(* PLC project Unnamed, Unknown Unnamed 1 *)
(* stored: creationDateTime 2025-10-24T15:36:12, modificationDateTime 2026-02-02T21:17:16 *)

PROGRAM program0
  VAR
    RawADC : INT;
    Temp : INT;
  END_VAR

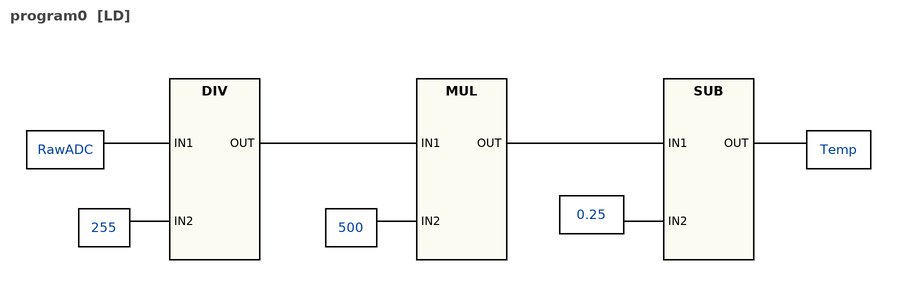
(* LD diagram, written out as Structured Text *)
Temp := RawADC / 255 * 500 - 0.25;
END_PROGRAM

CONFIGURATION Config0
  RESOURCE Res0 ON PLC
    TASK task0(INTERVAL := T#20ms, PRIORITY := 0);
    PROGRAM instance0 WITH task0 : program0;
  END_RESOURCE
END_CONFIGURATION
